(* Logix 5000 project; controller Program_Dampproduktion Emulate 5570 rev 32.11; software revision 32.02 *)

TASK MainTask (continuous, watchdog 500 ms) : Simulering

MODULES
   Local : Emulate 5570 (ICP 3, rev 32.11)
END_MODULES

ADD_ON_INSTRUCTION DampProces   (* revision 1.0, vendor JPJohansen  *)
// Til obligatorisk opgave 1 - PA3
// Revision note:
// ændringer på dødtid og tidskonstant samt navn. den
VAR_INPUT
   belastning : REAL;
   DeadTime : REAL := 2.0;   // Dødtid 0.1 til 1.99 sek.
   Tidskonstant : REAL := 20.0;   // Tidskonstant i LeadLag 0.1 til 40.0 sek
END_VAR
VAR_OUTPUT
   PV : REAL; {access Read Only, required}
END_VAR
VAR_INPUT
   CV : REAL; {required}
END_VAR
VAR
   DEDT_01 : DEADTIME := (Deadtime := 1.0, Gain := 1.0, RTSTime := 1);
   ADD_01 : FBD_MATH;
   LDLG_01 : LEAD_LAG := (Lag := 20.0, Gain := 1.0, RTSTime := 1);
   HLL_01 : HL_LIMIT := (HighLimit := 100.0);
   SCL_01 : SCALE := (InRawMax := 100.0, InEUMax := 15.0, Limiting := 1); {access None}
   SCL_02 : SCALE := (InRawMax := 100.0, InEUMax := -100.0, Limiting := 1); {access None}
   StorageA : REAL[200]; {access None}
   SCL_03 : SCALE := (InRawMax := 100.0, InEUMin := 100.0, Limiting := 1); {access None}
   __lBFE748FCFA657C66 : REAL; {access None}
   __l111F0F8E6DFC85BE : REAL; {access None}
END_VAR

ROUTINE Logic   (* function block diagram *)
   SHEET 1
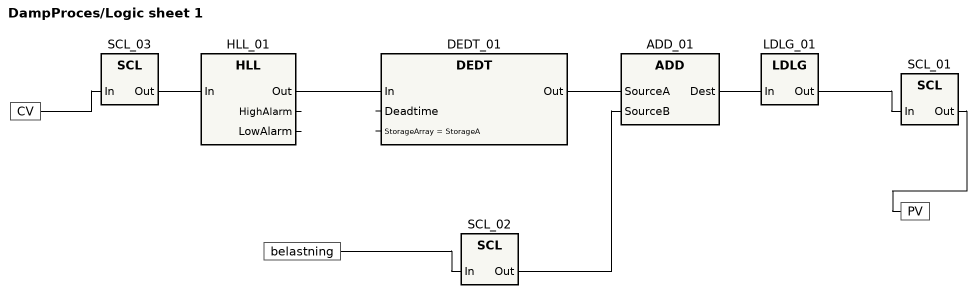
   SCL_03 : SCL(In := CV);
   HLL_01 : HLL(In := SCL_03.Out);   // unwired pins: HighAlarm LowAlarm
   DEDT_01 : DEDT(In := HLL_01.Out, StorageArray := StorageA);   // unwired pins: Deadtime
   SCL_02 : SCL(In := belastning);
   ADD_01 : ADD(SourceA := DEDT_01.Out, SourceB := SCL_02.Out);
   LDLG_01 : LDLG(In := ADD_01.Dest);
   SCL_01 : SCL(In := LDLG_01.Out);
   PV := SCL_01.Out;
END_ROUTINE
END_ADD_ON_INSTRUCTION

ADD_ON_INSTRUCTION Elektrodekammer   (* revision 1.0 *)
VAR_INPUT
   CV_Ind : REAL; {required}
END_VAR
VAR_OUTPUT
   PV_vandhojde : REAL; {access Read Only, required}
END_VAR
VAR_INPUT
   Belastning : REAL; {visible}
END_VAR
VAR
   LDLG_01 : LEAD_LAG := (Lag := 15.0, Gain := 1.4, RTSTime := 1); {access None}
   SUB_01 : FBD_MATH; {access None}
   DEDT_01 : DEADTIME := (Deadtime := 1.5, Gain := 1.5, RTSTime := 1); {access None}
   SCL_01 : SCALE := (InRawMax := 100.0, InEUMax := 100.0, Limiting := 1); {access None}
   SCL_02 : SCALE := (InRawMax := 100.0, InEUMax := 100.0, Limiting := 1); {access None}
   LDLG_02 : LEAD_LAG := (Lag := 10.0, Gain := 1.0, RTSTime := 1); {access None}
   Lag : REAL := 6.5; {access None}
   Gain_2 : REAL := 1.4; {access None}
   DeadTime : REAL := 0.5; {access None}
   Gain_1 : REAL := 0.9; {access None}
   StoreE : REAL[200]; {access None}
   __lBBB61524A4CF2047 : REAL; {access None}
   __l4C9B70D5358FCD80 : REAL; {access None}
   __lBCA77EE58B9857CC : REAL; {access None}
   __l311EF888CEB54C2F : REAL; {access None}
   __l26B57578D4CD21A6 : REAL; {access None}
   __l8BCF7D00DE459D5C : REAL; {access None}
END_VAR

ROUTINE Logic   (* function block diagram *)
   SHEET 1
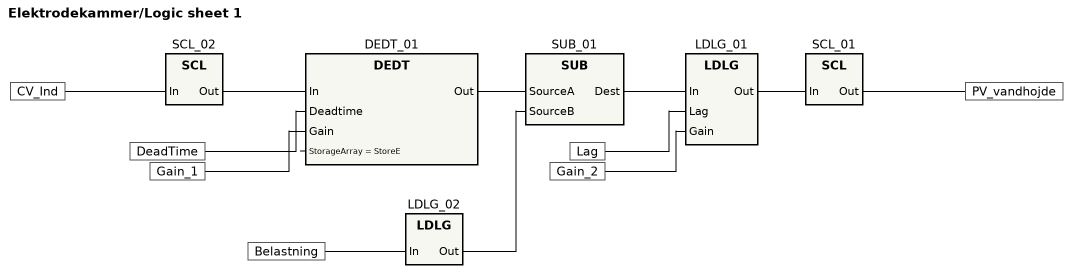
   SCL_02 : SCL(In := CV_Ind);
   DEDT_01 : DEDT(In := SCL_02.Out, Deadtime := DeadTime, Gain := Gain_1, StorageArray := StoreE);
   LDLG_02 : LDLG(In := Belastning);
   SUB_01 : SUB(SourceA := DEDT_01.Out, SourceB := LDLG_02.Out);
   LDLG_01 : LDLG(In := SUB_01.Dest, Lag := Lag, Gain := Gain_2);
   SCL_01 : SCL(In := LDLG_01.Out);
   PV_vandhojde := SCL_01.Out;
END_ROUTINE
END_ADD_ON_INSTRUCTION

ADD_ON_INSTRUCTION Foedevandskammer   (* revision 1.0 *)
VAR_INPUT
   CV_Ind : REAL; {required}
   Belastning : REAL; {visible}
END_VAR
VAR_OUTPUT
   PV_vandhojde : REAL; {access Read Only, required}
END_VAR
VAR
   LDLG_01 : LEAD_LAG := (Lag := 15.0, Gain := 1.4, RTSTime := 1); {access None}
   SUB_01 : FBD_MATH; {access None}
   DEDT_01 : DEADTIME := (Deadtime := 1.5, Gain := 1.5, RTSTime := 1); {access None}
   SCL_01 : SCALE := (InRawMax := 100.0, InEUMax := 100.0, Limiting := 1); {access None}
   SCL_02 : SCALE := (InRawMax := 100.0, InEUMax := 150.0, Limiting := 1); {access None}
   LDLG_02 : LEAD_LAG := (Lag := 10.0, Gain := 1.0, RTSTime := 1); {access None}
   DeadTime : REAL := 1.0; {access None}
   Gain_1 : REAL := 1.1; {access None}
   Lag : REAL := 8.0; {access None}
   Gain_2 : REAL := 1.2; {access None}
   StoreF : REAL[200]; {access None}
   __l47B9F860FB7F34CC : REAL; {access None}
   __lBCEEC7B2562564CC : REAL; {access None}
   __l8BD366BFA30A9B21 : REAL; {access None}
   __l726FB40F300CE841 : REAL; {access None}
   __l213C2E7ECA7368D6 : REAL; {access None}
   __l53F5B97CD43989B2 : REAL; {access None}
END_VAR

ROUTINE Logic   (* function block diagram *)
   SHEET 1
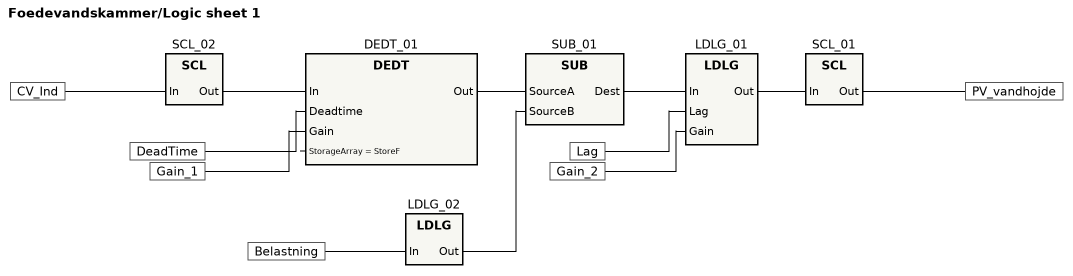
   SCL_02 : SCL(In := CV_Ind);
   DEDT_01 : DEDT(In := SCL_02.Out, Deadtime := DeadTime, Gain := Gain_1, StorageArray := StoreF);
   LDLG_02 : LDLG(In := Belastning);
   SUB_01 : SUB(SourceA := DEDT_01.Out, SourceB := LDLG_02.Out);
   LDLG_01 : LDLG(In := SUB_01.Dest, Lag := Lag, Gain := Gain_2);
   SCL_01 : SCL(In := LDLG_01.Out);
   PV_vandhojde := SCL_01.Out;
END_ROUTINE
END_ADD_ON_INSTRUCTION

ADD_ON_INSTRUCTION Kondenstank   (* revision 1.0, vendor Mr.Helgason *)
// Simulering af et kondenstank
// Help:
// *********************************
// Simulering af Vandmodeller
// *********************************
// Input:
// CV_in =  CV (Control Value) fra regulator 0-100% . REAL
// Belastning = Bruger indstiller 0 - 100%.  REAL
// Output:
// PV_vandhojde = Fra Level transmitter 0-100%. REAL
VAR_INPUT
   Belastning : REAL; {required}   // Belasting 0 - 100%
   CV_Ind : REAL; {required}   // 0 - 100%
END_VAR
VAR_OUTPUT
   PV_vandhojde : REAL; {access Read Only, required}   // 0 - 100%
END_VAR
VAR
   LDLG_01 : LEAD_LAG := (Lag := 15.0, Gain := 1.4, RTSTime := 1); {access None}
   SUB_01 : FBD_MATH; {access None}
   DEDT_01 : DEADTIME := (Deadtime := 1.5, Gain := 1.5, RTSTime := 1); {access None}
   DeadTime : REAL := 2.0; {access None}
   Store : REAL[200]; {access None}
   SCL_01 : SCALE := (InRawMax := 100.0, InEUMax := 100.0, Limiting := 1); {access None}
   SCL_02 : SCALE := (InRawMax := 100.0, InEUMax := 150.0, Limiting := 1); {access None}
   Gain_1 : REAL := 1.4; {access None}
   Lag : REAL := 15.0; {access None}
   Gain_2 : REAL := 1.2; {access None}
   LDLG_02 : LEAD_LAG := (Lag := 10.0, Gain := 1.0, RTSTime := 1); {access None}
   __l770FDFE62A3820F0 : REAL; {access None}
   __l2251F834FE043185 : REAL; {access None}
   __l3FFF9E27A9364976 : REAL; {access None}
   __lB3381F195010FDBE : REAL; {access None}
   __lEBAC3B9CE4C94A7F : REAL; {access None}
   __l23F97D3D6AB6734A : REAL; {access None}
END_VAR

ROUTINE Logic   (* function block diagram *)
   SHEET 1
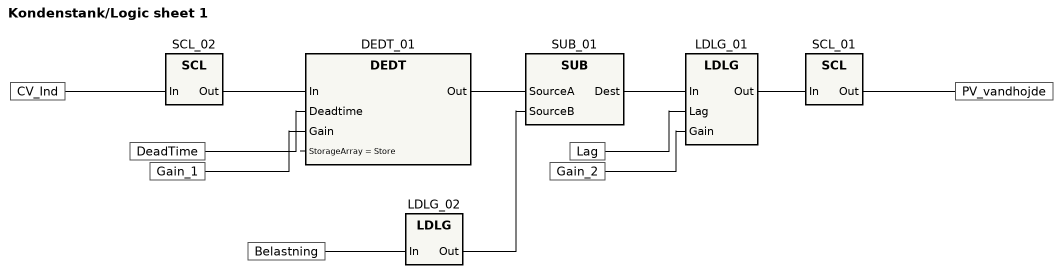
   SCL_02 : SCL(In := CV_Ind);
   DEDT_01 : DEDT(In := SCL_02.Out, Deadtime := DeadTime, Gain := Gain_1, StorageArray := Store);
   LDLG_02 : LDLG(In := Belastning);
   SUB_01 : SUB(SourceA := DEDT_01.Out, SourceB := LDLG_02.Out);
   LDLG_01 : LDLG(In := SUB_01.Dest, Lag := Lag, Gain := Gain_2);
   SCL_01 : SCL(In := LDLG_01.Out);
   PV_vandhojde := SCL_01.Out;
END_ROUTINE
END_ADD_ON_INSTRUCTION

VAR_GLOBAL   (* controller tags *)
   E1_E2 : BOOL;
   initialize : BOOL;
   initValue : REAL;
   Kd : REAL;
   Ki : REAL;
   PT_3 : REAL;
   SP : REAL;
   V3 : REAL;
END_VAR

PROGRAM Simulering   (* main routine DampProces_Simulering *)
VAR
   ADD_01 : FBD_MATH;
   DampProces_01 : DampProces := (DeadTime := 2.0, Tidskonstant := 20.0);
   INTG_01 : INTEGRATOR := (RTSTime := 1);
   MUL_01 : FBD_MATH;
   SUB_01 : FBD_MATH;
END_VAR

ROUTINE DampProces_Simulering   (* function block diagram *)
   SHEET 1
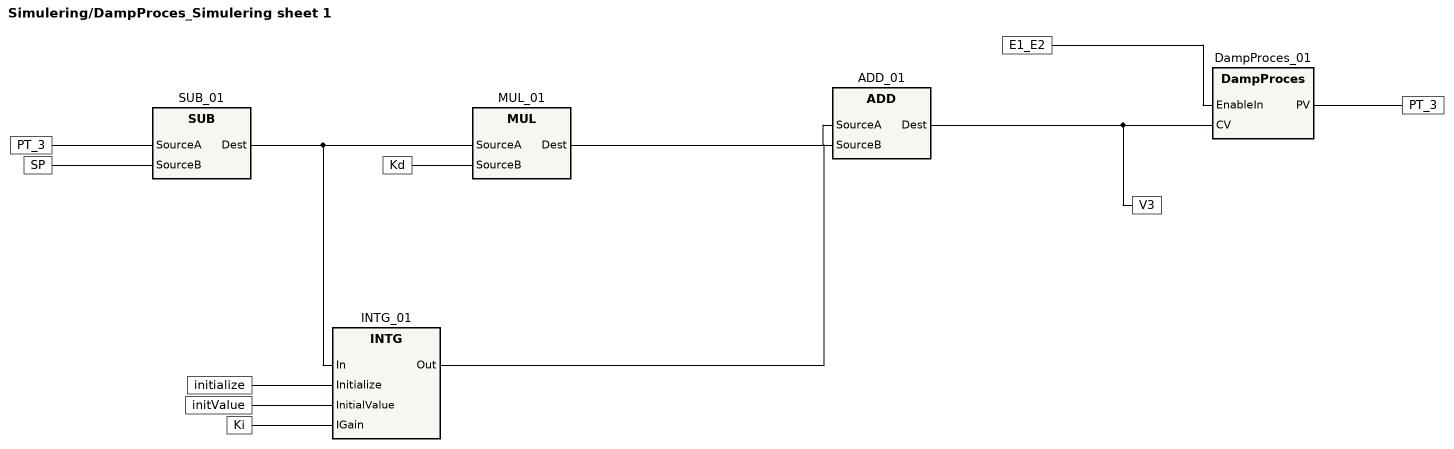
   SUB_01 : SUB(SourceA := PT_3, SourceB := SP);
   INTG_01 : INTG(In := SUB_01.Dest, Initialize := initialize, InitialValue := initValue, IGain := Ki);
   MUL_01 : MUL(SourceA := SUB_01.Dest, SourceB := Kd);
   ADD_01 : ADD(SourceA := MUL_01.Dest, SourceB := INTG_01.Out);
   V3 := ADD_01.Dest;
   DampProces_01 : DampProces(EnableIn := E1_E2, CV := ADD_01.Dest);
   PT_3 := DampProces_01.PV;
END_ROUTINE
END_PROGRAM
